(* PLC project Unnamed, Unknown Unnamed 1 *)
(* stored: creationDateTime 2026-05-29T19:35:44, modificationDateTime 2026-05-29T19:35:44 *)

PROGRAM main
  VAR
    Q_READY AT %QX0.0 : BOOL := False;
    Q_REQUEST AT %QX0.1 : BOOL := False;
    Q_PASS_ALLOWED AT %QX0.2 : BOOL := False;
    Q_EMERGENCY AT %QX0.3 : BOOL := False;
    CMD_ROBOT_REQUEST AT %QX80.0 : BOOL := False;
    CMD_HMI_ALLOW AT %QX80.1 : BOOL := False;
    CMD_ROBOT_PASSED AT %QX80.2 : BOOL := False;
    CMD_EMERGENCY AT %QX80.3 : BOOL := False;
    CMD_RESET AT %QX80.4 : BOOL := False;
    STATUS_READY AT %QX81.0 : BOOL := False;
    STATUS_REQUEST AT %QX81.1 : BOOL := False;
    STATUS_PASS_ALLOWED AT %QX81.2 : BOOL := False;
    STATUS_EMERGENCY AT %QX81.3 : BOOL := False;
    STATUS_BARRIER_OPEN AT %QX81.4 : BOOL := False;
    STATUS_PASS_PERMISSION AT %QX81.5 : BOOL := False;
  END_VAR
  VAR
    M_READY : BOOL := True;
    M_REQUEST : BOOL := False;
    M_PASS_ALLOWED : BOOL := False;
    M_EMERGENCY : BOOL := False;
    STA : BOOL;
  END_VAR

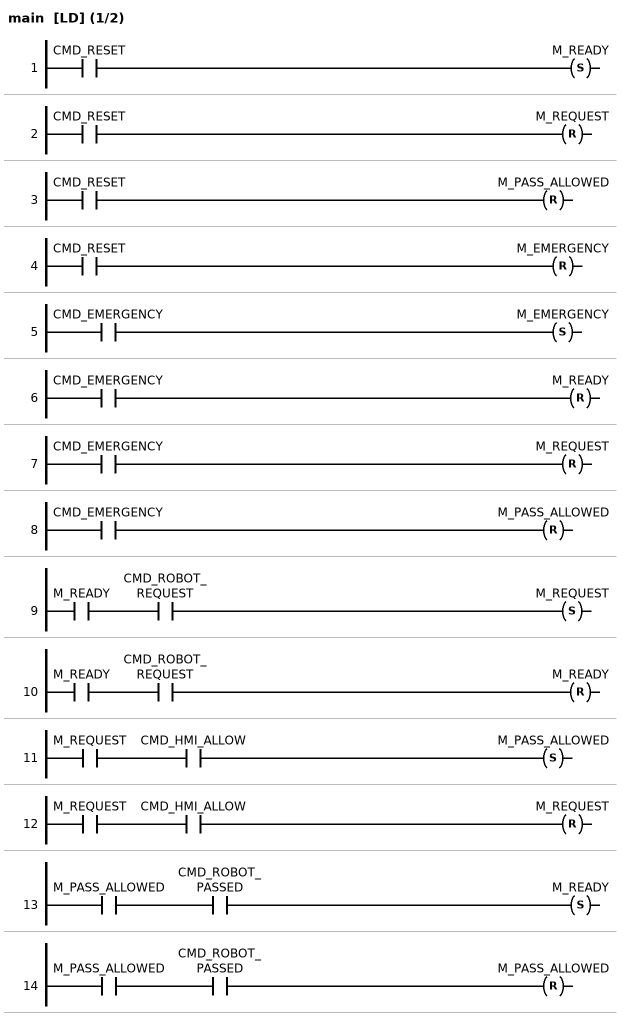
(* LD diagram, written out as Structured Text *)
IF CMD_RESET THEN M_READY := TRUE; END_IF;
IF CMD_RESET THEN M_REQUEST := FALSE; END_IF;
IF CMD_RESET THEN M_PASS_ALLOWED := FALSE; END_IF;
IF CMD_RESET THEN M_EMERGENCY := FALSE; END_IF;
IF CMD_EMERGENCY THEN M_EMERGENCY := TRUE; END_IF;
IF CMD_EMERGENCY THEN M_READY := FALSE; END_IF;
IF CMD_EMERGENCY THEN M_REQUEST := FALSE; END_IF;
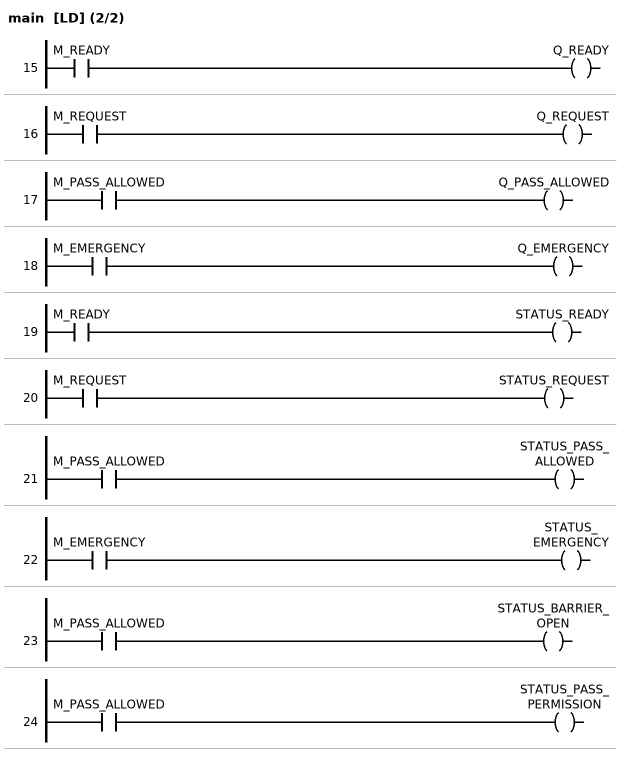
IF CMD_EMERGENCY THEN M_PASS_ALLOWED := FALSE; END_IF;
IF M_READY AND CMD_ROBOT_REQUEST THEN M_REQUEST := TRUE; END_IF;
IF M_READY AND CMD_ROBOT_REQUEST THEN M_READY := FALSE; END_IF;
IF M_REQUEST AND CMD_HMI_ALLOW THEN M_PASS_ALLOWED := TRUE; END_IF;
IF M_REQUEST AND CMD_HMI_ALLOW THEN M_REQUEST := FALSE; END_IF;
IF M_PASS_ALLOWED AND CMD_ROBOT_PASSED THEN M_READY := TRUE; END_IF;
IF M_PASS_ALLOWED AND CMD_ROBOT_PASSED THEN M_PASS_ALLOWED := FALSE; END_IF;
Q_READY := M_READY;
Q_REQUEST := M_REQUEST;
Q_PASS_ALLOWED := M_PASS_ALLOWED;
Q_EMERGENCY := M_EMERGENCY;
STATUS_READY := M_READY;
STATUS_REQUEST := M_REQUEST;
STATUS_PASS_ALLOWED := M_PASS_ALLOWED;
STATUS_EMERGENCY := M_EMERGENCY;
STATUS_BARRIER_OPEN := M_PASS_ALLOWED;
STATUS_PASS_PERMISSION := M_PASS_ALLOWED;
END_PROGRAM

CONFIGURATION Config0
  RESOURCE Res0 ON PLC
    TASK task0(INTERVAL := T#20ms, PRIORITY := 1);
    PROGRAM instance0 WITH task0 : main;
  END_RESOURCE
END_CONFIGURATION
